// TwinCAT 3 PLC project Example
// ProgramVersion: 3.1.4026.19
// libraries:
//   Bolt, * (Zeugwerk GmbH)
//   Struckig, 0.15.5.0 (Stefan Besler)
//   Tc3_Module, * (Beckhoff Automation GmbH)
//   ZApplication, 1.5.37.1 (Zeugwerk GmbH)
//   ZAux, 1.5.37.1 (Zeugwerk GmbH)
//   ZCore, 1.5.37.1 (Zeugwerk GmbH)
//   ZEquipment, 1.5.37.1 (Zeugwerk GmbH)
//   ZPlatform, 1.5.37.1 (Zeugwerk GmbH)
// project tree:
//   ZApp/App/ ZApp.TcPOU
//   ZApp/App/_DataTypes/ ZAppStep.TcDUT
//   ZApp/App/_States/ ZAppSequenceBoot.TcPOU, ZAppSequenceBootFault.TcPOU, ZAppSequenceRunning.TcPOU
//   ZApp/App/_SubObjects/ ZAppSequence.TcPOU
//   ZApp/Com/_DataTypes/ ZCom.TcDUT (not stored), ZComUnit.TcDUT
//   ZApp/Data/_DataTypes/ ZData.TcDUT, ZDataMachine.TcDUT, ZDataConfig.TcDUT, ZDataCalibration.TcDUT (not stored), ZDataRecipe.TcDUT (not stored)
//   ZApp/Unit/Handling/ HandlingUnit.TcPOU, HandlingUnitProgram.TcPOU, IHandling.TcIO (not stored)
//   ZApp/Unit/Handling/_Com/ HandlingCom.TcDUT (not stored), HandlingComPublish.TcDUT (not stored), HandlingComPublishEquipment.TcDUT (not stored), HandlingComRef.TcDUT, HandlingComRequest.TcDUT (not stored), HandlingComSubscribe.TcDUT, HandlingComSubscribeEquipment.TcDUT (not stored)
//   ZApp/Unit/Handling/_DataTypes/ HandlingState.TcDUT, HandlingStep.TcDUT
//   ZApp/Unit/Handling/_Data/ HandlingDataCalibration.TcDUT (not stored), HandlingDataConfig.TcDUT, HandlingDataMachine.TcDUT, HandlingDataRef.TcDUT
//   ZApp/Unit/Handling/_Equipment/ HandlingActuator.TcPOU, HandlingAxis.TcPOU (not stored), HandlingCollision.TcPOU, HandlingEquipment.TcPOU (not stored), HandlingFieldbus.TcPOU (not stored), HandlingIo.TcPOU, HandlingLinkedUnit.TcPOU
//   ZApp/Unit/Handling/_States/ HandlingSequenceAutomatic.TcPOU, HandlingSequenceBoot.TcPOU, HandlingSequenceFaultReaction.TcPOU (not stored), HandlingSequenceGoHome.TcPOU (not stored), HandlingSequenceStop.TcPOU
//   ZApp/Unit/Handling/_SubObjects/ HandlingContainer.TcPOU, HandlingSequence.TcPOU
//   ZApp/Unit/Mover/ IMover.TcIO (not stored), MoverUnit.TcPOU, MoverUnitProgram.TcPOU
//   ZApp/Unit/Mover/_Com/ MoverCom.TcDUT, MoverComPublish.TcDUT (not stored), MoverComPublishEquipment.TcDUT, MoverComRef.TcDUT, MoverComRequest.TcDUT (not stored), MoverComSubscribe.TcDUT (not stored), MoverComSubscribeEquipment.TcDUT
//   ZApp/Unit/Mover/_DataTypes/ MoverState.TcDUT, MoverStep.TcDUT (not stored)
//   ZApp/Unit/Mover/_Data/ MoverDataCalibration.TcDUT (not stored), MoverDataConfig.TcDUT (not stored), MoverDataMachine.TcDUT (not stored), MoverDataRef.TcDUT
//   ZApp/Unit/Mover/_Equipment/ MoverCollision.TcPOU (not stored), MoverActuator.TcPOU, MoverAxis.TcPOU (not stored), MoverEquipment.TcPOU (not stored), MoverFieldbus.TcPOU (not stored), MoverIo.TcPOU, MoverLinkedUnit.TcPOU
//   ZApp/Unit/Mover/_States/ MoverSequenceAutomatic.TcPOU (not stored), MoverSequenceBoot.TcPOU, MoverSequenceFaultReaction.TcPOU (not stored), MoverSequenceGoHome.TcPOU (not stored), MoverSequenceStop.TcPOU (not stored)
//   ZApp/Unit/Mover/_SubObjects/ MoverContainer.TcPOU, MoverSequence.TcPOU (not stored)
//   ZApp/ ZGlobal.TcGVL (not stored), ZModuleProgram.TcPOU, ZModuleTask.TcTTO (not stored)
// real-time tasks:
//   TASK ZModuleTask: cycle T#10ms, priority 20, ADS port 350

// ---- ZApp/App/_DataTypes/ZAppStep.TcDUT
{attribute 'qualified_only'}
{attribute 'to_string'}
TYPE ZAppStep :
(
  Undefined := 0
  
  ,BootBegin
  ,BootLoadDefaultData
  ,BootEnd
  ,BootFaultBegin
  ,BootFaultEnd 
  ,RunningBegin
  ,RunningEnd   
);
END_TYPE

// ---- ZApp/Com/_DataTypes/ZComUnit.TcDUT
TYPE ZComUnit :
STRUCT
{region "Handling"}
{IF NOT (defined (Handling_disabled))}
  Handling : HandlingCom;
  {attribute 'ZId' := 'a0dd13f9-743a-4c3b-9b43-ecc916834d10'}
{END_IF}
{endregion}
{region "Mover1"}
{IF NOT (defined (Mover1_disabled))}
  Mover1 : MoverCom;
  {attribute 'ZId' := '0635b537-20e6-40de-ab4b-39921311b510'}
{END_IF}
{endregion}
{attribute '__ZwPlcApplicationComUnitDeclaration__'} // Do not remove this attribute! It is used for code generation.
END_STRUCT
END_TYPE

// ---- ZApp/Data/_DataTypes/ZData.TcDUT
TYPE ZData :
STRUCT
  Config : ZDataConfig;
  Machine : ZDataMachine;
  Calibration : ZDataCalibration;
  Recipe : ZDataRecipe;
END_STRUCT
END_TYPE

// ---- ZApp/Data/_DataTypes/ZDataMachine.TcDUT
TYPE ZDataMachine :
STRUCT
{region "Handling"}
{IF NOT (defined (Handling_disabled))}
  Handling : HandlingDataMachine;
  {attribute 'ZId' := 'a0dd13f9-743a-4c3b-9b43-ecc916834d10'}
{END_IF}
{endregion}
{region "Mover1"}
{IF NOT (defined (Mover1_disabled))}
  Mover1 : MoverDataMachine;
  {attribute 'ZId' := '0635b537-20e6-40de-ab4b-39921311b510'}
{END_IF}
{endregion}
{attribute '__ZwPlcApplicationDataMachineDeclaration__'} // Do not remove this attribute! It is used for code generation.
END_STRUCT
END_TYPE

// ---- ZApp/Data/_DataTypes/ZDataConfig.TcDUT
TYPE ZDataConfig :
STRUCT
{region "Handling"}
{IF NOT (defined (Handling_disabled))}
  Handling : HandlingDataConfig;
  {attribute 'ZId' := 'a0dd13f9-743a-4c3b-9b43-ecc916834d10'}
{END_IF}
{endregion}
{region "Mover1"}
{IF NOT (defined (Mover1_disabled))}
  Mover1 : MoverDataConfig;
  {attribute 'ZId' := '0635b537-20e6-40de-ab4b-39921311b510'}
{END_IF}
{endregion}
{attribute '__ZwPlcApplicationDataConfigDeclaration__'} // Do not remove this attribute! It is used for code generation.
END_STRUCT
END_TYPE

// ---- ZApp/Unit/Handling/_Com/HandlingComRef.TcDUT
/// container for all communication data types that are used by the unit
TYPE HandlingComRef :
STRUCT
  Publish : REFERENCE TO HandlingComPublish; 
  Subscribe : REFERENCE TO HandlingComSubscribe; 
END_STRUCT
END_TYPE

// ---- ZApp/Unit/Handling/_Com/HandlingComSubscribe.TcDUT
TYPE HandlingComSubscribe :
STRUCT
  Request : HandlingComRequest; // contains booleans that are used to start a specific sequence.
  Equipment : HandlingComSubscribeEquipment;  // structs for equipment objects which are used by the bridges
END_STRUCT
END_TYPE

// ---- ZApp/Unit/Handling/_DataTypes/HandlingState.TcDUT
/// This enumeration contains all used defined sequences of a unit.
/// Per default a unit makes use of the states that are contained in (UnitStateDefault)[xref:ZApplication.UnitStateDefault]. However,
/// most of the time a unit need to perform some application depend sequences that can be performed by putting the unit into userdefined states.
/// For instance, a robotic unit could use the state (automatic)[xref:ZApplication.UnitStateDefault] to lift an object from point A to point B,
/// a userdefined state could be used to open and close the robotic-units gripper, respectively
{attribute 'qualified_only'}
TYPE HandlingState :
(
	UserdefinedState1 := ZApplication.UnitStateMachineState.Last+1
);
END_TYPE

// ---- ZApp/Unit/Handling/_DataTypes/HandlingStep.TcDUT
/// This enumeration contains all steps that are used by the various sequences of a unit.
/// Sequences use a subrange (***Begin to ***End) of this enumeration.
{attribute 'qualified_only'}
{attribute 'to_string'}
TYPE HandlingStep :
(
  Undefined := 0
  
  ,BootBegin
  ,BootEnd 

  ,StopBegin
  ,StopEnd

  ,AutomaticBegin
  ,AutomaticSwitch
  ,AutomaticMoveInterpolatedVelocity
  ,AutomaticEnd
  
  ,GoHomeBegin
  ,GoHomeJoint3
  ,GoHomeJoint12
  ,GoHomeJoint2
  ,GoHomeEnd 
  
  ,FaultReactionBegin
  ,FaultReactionEnd
);
END_TYPE

// ---- ZApp/Unit/Handling/_Data/HandlingDataConfig.TcDUT
/// configuration data that is used during boot to configure the Units equipment
TYPE HandlingDataConfig :
STRUCT
  Simulated : BOOL;
END_STRUCT
END_TYPE

// ---- ZApp/Unit/Handling/_Data/HandlingDataMachine.TcDUT
/// machine data that is used through most sequences of the unit (motor speed, axes positions, ...)
TYPE HandlingDataMachine :
STRUCT
  Slowspeed : LREAL;
  Highspeed : LREAL;
END_STRUCT
END_TYPE

// ---- ZApp/Unit/Handling/_Data/HandlingDataRef.TcDUT
/// container for all data that are used by the unit
TYPE HandlingDataRef :
STRUCT
  Config : REFERENCE TO HandlingDataConfig; // data required for booting the unit (axes configuration, simulation, parameters that have to be written in PREOP, ...)
  Machine : REFERENCE TO HandlingDataMachine; // speeds, positions, ...
  Calibration : REFERENCE TO HandlingDataCalibration; // offsets, shifts of nominal to actual values
END_STRUCT
END_TYPE

// ---- ZApp/Unit/Mover/_Com/MoverCom.TcDUT
/// This struct contains variables that
/// * are read from outside (e.g. HMI) to retrieve information about the unit's current state and (temporary) parameters (= `publish`) 
/// * are written from outside (e.g. HMI) to control the unit via ADS (= `subscribe`) 
TYPE MoverCom :
STRUCT
  Publish : MoverComPublish;
  Subscribe : MoverComSubscribe;
END_STRUCT
END_TYPE

// ---- ZApp/Unit/Mover/_Com/MoverComPublishEquipment.TcDUT
TYPE MoverComPublishEquipment :
STRUCT

{region "AxisX : Axis"}
  AxisX : ZApplication.AxisComPublish;
  {attribute 'ZId' := '002e5115-61f4-40c1-8715-993ad81c0703'}
{endregion}

{attribute '__ZwPlcUnitComDeclaration__'} // Do not remove this attribute! It is used for code generation.

END_STRUCT
END_TYPE

// ---- ZApp/Unit/Mover/_Com/MoverComRef.TcDUT
/// container for all communication data types that are used by the unit
TYPE MoverComRef :
STRUCT
  Publish : REFERENCE TO MoverComPublish; 
  Subscribe : REFERENCE TO MoverComSubscribe; 
END_STRUCT
END_TYPE

// ---- ZApp/Unit/Mover/_Com/MoverComSubscribeEquipment.TcDUT
TYPE MoverComSubscribeEquipment :
STRUCT

{region "AxisX : Axis"}
  AxisX : ZApplication.AxisComSubscribe;
  {attribute 'ZId' := '002e5115-61f4-40c1-8715-993ad81c0703'}
{endregion}

{attribute '__ZwPlcUnitComDeclaration__'} // Do not remove this attribute! It is used for code generation.

END_STRUCT
END_TYPE

// ---- ZApp/Unit/Mover/_DataTypes/MoverState.TcDUT
/// This enumeration contains all used defined sequences of a unit.
/// Per default a unit makes use of the states that are contained in (UnitStateDefault)[xref:ZApplication.UnitStateDefault]. However,
/// most of the time a unit need to perform some application depend sequences that can be performed by putting the unit into userdefined states.
/// For instance, a robotic unit could use the state (automatic)[xref:ZApplication.UnitStateDefault] to lift an object from point A to point B,
/// a userdefined state could be used to open and close the robotic-units gripper, respectively
{attribute 'qualified_only'}
TYPE MoverState :
(
	UserdefinedState1 := ZApplication.UnitStateMachineState.Last+1
);
END_TYPE

// ---- ZApp/Unit/Mover/_Data/MoverDataRef.TcDUT
/// container for all data that are used by the unit
TYPE MoverDataRef :
STRUCT
  Config : REFERENCE TO MoverDataConfig; // data required for booting the unit (axes configuration, simulation, parameters that have to be written in PREOP, ...)
  Machine : REFERENCE TO MoverDataMachine; // speeds, positions, ...
  Calibration : REFERENCE TO MoverDataCalibration; // offsets, shifts of nominal to actual values
END_STRUCT
END_TYPE

// ---- ZApp/App/ZApp.TcPOU
FUNCTION_BLOCK ZApp EXTENDS ZApplication.Application
VAR
  _boot : ZAppSequenceBoot;
  _bootFault : ZAppSequenceBootFault;
  _running : ZAppSequenceRunning;
END_VAR

METHOD FB_init : BOOL
VAR_INPUT
  bInitRetains : BOOL; /// if TRUE, the retain variables are initialized (warm start / cold start)
  bInCopyCode : BOOL; /// if TRUE, the instance afterwards gets moved into the copy code (online change)
  displayName : ZCore.ZString;
  com : REFERENCE TO ZApplication.ApplicationComPublish;
END_VAR
SetBootSequence(_boot);
SetBootFaultSequence(_bootFault);
SetRunningSequence(_running);
END_METHOD

END_FUNCTION_BLOCK

// ---- ZApp/App/_States/ZAppSequenceBoot.TcPOU
FUNCTION_BLOCK ZAppSequenceBoot EXTENDS ZAppSequence IMPLEMENTS ZCore.ISequence
VAR
  _step : ZCore.Step(ZAppStep.BootBegin, ZAppStep.BootEnd);
END_VAR

IF OnStart(_step)
THEN
  // init custom sequence variables here ...
END_IF

REPEAT
  LogStep();

  CASE _step.Index OF
    (* -------------------------------------------------------------------------------------------------------------------------------- *)
    ZAppStep.BootBegin:
    (* -------------------------------------------------------------------------------------------------------------------------------- *)
    
      IF _step.OnEntry()
      THEN
        ZModuleProgram.LoggerFile.MinimumLevel := ZCore.LogLevel.Trace;
        ZModuleProgram.Logger.AddLogger(ZModuleProgram.LoggerFile); 
        //ZModuleProgram.World.Host := '82.165.219.190.1.1';       
        ZModuleProgram.World.SetLogger(ZModuleProgram.Logger);
        {attribute '__ZwPlcAppZComModuleContext__'} // Do not remove this attribute! It is used for code generation.      
      END_IF
      
	  IF ZModuleProgram.Datetime.State <> ZCore.ObjectState.Booting
      THEN
        _step.SetNext(ZAppStep.BootLoadDefaultData);        
      END_IF
      
    (* -------------------------------------------------------------------------------------------------------------------------------- *)
    ZAppStep.BootLoadDefaultData:
    (* -------------------------------------------------------------------------------------------------------------------------------- *)

      {warning 'The application is loading the default config data on every restart!'}
      LoadDefaultConfigData();
      
      IF IsCommissioning()
      THEN
        LoadDefaultData();
      END_IF
      
      _step.SetNext(ZAppStep.BootEnd);
      
    (* -------------------------------------------------------------------------------------------------------------------------------- *)
    ZAppStep.BootEnd:
    (* -------------------------------------------------------------------------------------------------------------------------------- *)
      SetBusy(FALSE);
      
  ELSE
    Abort('sequence contains unhandled step');
  END_CASE
UNTIL _step.IsNotRepeatable() OR_ELSE NOT Busy END_REPEAT

METHOD  IsCommissioning : BOOL
IsCommissioning := TRUE;
END_METHOD

METHOD FINAL LoadDefaultConfigData

{region "Handling"}
  {IF NOT (defined (Handling_disabled))}
  ZGlobal.Data.Config.Handling.Simulated := TRUE;
  {region "UserInitCode"}
  // put your individual init code for this unit here
  {endregion}
  {END_IF}
  {attribute 'ZId' := 'a0dd13f9-743a-4c3b-9b43-ecc916834d10'}
{endregion}

{region "Mover1"}
  {IF NOT (defined (Mover1_disabled))}
  ZGlobal.Data.Config.Mover1.Simulated := TRUE;
  {region "UserInitCode"}
  // put your individual init code for this unit here
  {endregion}
  {END_IF}
  {attribute 'ZId' := '0635b537-20e6-40de-ab4b-39921311b510'}
{endregion}

{attribute '__ZwPlcUnitLoadDefaultConfigData__'} // Do not remove this attribute! It is used for code generation.
END_METHOD

METHOD FINAL LoadDefaultData

{attribute '__ZwPlcUnitLoadDefaultData__'} // Do not remove this attribute! It is used for code generation.
END_METHOD

END_FUNCTION_BLOCK

// ---- ZApp/App/_SubObjects/ZAppSequence.TcPOU
FUNCTION_BLOCK ABSTRACT ZAppSequence EXTENDS ZApplication.Sequence IMPLEMENTS ZCore.ISequence

METHOD StepDecoded : ZCore.ZString
VAR_INPUT
  stepIndex : INT;
END_VAR
VAR_INST
  _stepIndexDecoded : ZAppStep;
END_VAR
_stepIndexDecoded := stepIndex;
StepDecoded := TO_STRING(_stepIndexDecoded);
END_METHOD

END_FUNCTION_BLOCK

// ---- ZApp/ZModuleProgram.TcPOU
/// Zeugwerk Application
PROGRAM ZModuleProgram
VAR_INPUT
{region "ZModuleProgram : Utility"}
  App : ZApp(displayName:='Zeugwerk-Application Template', com:=ZGlobal.Com.App);
  Datetime : ZAux.DateTimeUM;
  {attribute 'ZId' := ''}
{endregion}
{region "ZModuleProgram : Logging"}
  Alarming : ZApplication.Alarming(App, datetime := Datetime, com := ZGlobal.Com.Alarming);
  LoggerHmi : ZApplication.Messaging(App, datetime := Datetime, com := ZGlobal.Com.Messages);
  LoggerFile : ZAux.LoggerFile7FF(App, datetime := Datetime, filePath:='C:\Zeugwerk\logs\messages.log', target:='');
  Logger : ZAux.Logging;
  World : Bolt.CollisionWorld(App, 'E:\Bullcat\Example\world.urdf');
  {attribute 'ZId' := ''}
{endregion}  
{attribute '__ZwPlcApplicationModuleProgramDeclaration__'} // Do not remove this attribute! It is used for code generation.
{region "Handling"}
{undefine RunInSeparateProgram}
{IF NOT (defined (Handling_disabled)) AND NOT (defined (RunInSeparateProgram))}
  Handling : HandlingUnit(displayName := 'Handling', // name of the unit (for logging)
					  parent := App, // caller of the Unit's cyclic method. If the Unit runs in its own context use 0
						configdata := ZGlobal.Data.Config.Handling,
						machinedata := ZGlobal.Data.Machine.Handling,
						calibrationdata := ZGlobal.Data.Calibration.Handling,
						com := ZGlobal.Com.Unit.Handling);
  {attribute 'section' := '__ZwPlcUnitProgramDeclaration__'}
  {attribute 'ZId' := 'a0dd13f9-743a-4c3b-9b43-ecc916834d10'}
{END_IF}
{endregion}
{region "Mover1"}
{undefine RunInSeparateProgram}
{IF NOT (defined (Mover1_disabled)) AND NOT (defined (RunInSeparateProgram))}
  Mover1 : MoverUnit(displayName := 'Mover1', // name of the unit (for logging)
    parent:= App,
    configdata:= ZGlobal.Data.Config.Mover1,
    machinedata := ZGlobal.Data.Machine.Mover1,
    calibrationdata := ZGlobal.Data.Calibration.Mover1,
    com := ZGlobal.Com.Unit.Mover1,
    logger := Logger,
    alarming:= Alarming);
  {attribute 'section' := '__ZwPlcUnitProgramDeclaration__'}
  {attribute 'ZId' := '0635b537-20e6-40de-ab4b-39921311b510'}
{END_IF}
{endregion}
{attribute '__ZwPlcUnitProgramDeclaration__'} // Do not remove this attribute! It is used for code generation.
END_VAR

// do collision detection for whole machine
IF NOT World.Busy
THEN
  World.UpdateAndCheckSceneAsync();
END_IF

{region "ZModuleProgram : Utility"}
  Datetime.Cyclic();
  App.Cyclic();
  {attribute 'ZId' := ''}
{endregion}
{attribute '__ZwPlcApplicationModuleProgramImplementation__'} // Do not remove this attribute! It is used for code generation.

END_PROGRAM

// ---- ZApp/Unit/Handling/HandlingUnit.TcPOU
/// Declaration of a distinct unit of this application
FUNCTION_BLOCK HandlingUnit EXTENDS ZApplication.Unit IMPLEMENTS IHandling
VAR
  _equipment : HandlingEquipment(THIS^);
  _data : HandlingDataRef;
  _com : HandlingComRef;

  _boot : HandlingSequenceBoot(THIS^);
  _automatic : HandlingSequenceAutomatic(THIS^);
  _stop : HandlingSequenceStop(THIS^);
  _gohome : HandlingSequenceGoHome(THIS^);
  _faultReaction : HandlingSequenceFaultReaction(THIS^);
  
  _statemachine : ZApplication.UnitStateMachine;

  _observeTimer : ZAux.Timer;
END_VAR

{attribute 'ZId' := '2160a0d9-b961-4504-830a-bd7771ead3e7'}

IF _observeTimer.Done THEN
  _observeTimer.WaitAsync(0.1);
  
  // monitor _com for requested actions (e.g. start homing, start automatic mode, ...)
  ObserveRequest(_com.Subscribe.Request.Start, ZApplication.UnitStateMachineState.Automatic);
  ObserveRequest(_com.Subscribe.Request.Stop, ZApplication.UnitStateMachineState.Stop);
  ObserveRequest(_com.Subscribe.Request.GoHome, ZApplication.UnitStateMachineState.GoHome);
  ObserveRequest(_com.Subscribe.Request.Halt, ZApplication.UnitStateMachineState.Halt);
  
  // provide relevant information via ADS
  _com.Publish.Request.Stop := _stateMachine.IsTransitionAllowed(ZApplication.UnitStateMachineState.Stop);
  _com.Publish.Request.Start := _stateMachine.IsTransitionAllowed(ZApplication.UnitStateMachineState.Automatic);
  _com.Publish.Request.GoHome := _stateMachine.IsTransitionAllowed(ZApplication.UnitStateMachineState.GoHome);
  _com.Publish.Request.Halt := _stateMachine.IsTransitionAllowed(ZApplication.UnitStateMachineState.Halt);

  _com.Publish.State := _stateMachine.State();
END_IF

IF _statemachine.State() <> UnitStateMachineState.Automatic
THEN
  _equipment.Collision.Joint1.SetPosition((_equipment.Axis.Axis1.ActualPosition + _equipment.Axis.Axis1.ActualFollowingError) / 180.0 * ZCore.Constants.Pi);
  _equipment.Collision.Joint2.SetPosition((_equipment.Axis.Axis2.ActualPosition + _equipment.Axis.Axis2.ActualFollowingError) / 180.0 * ZCore.Constants.Pi);
  _equipment.Collision.Joint3.SetPosition((_equipment.Axis.Axis3.ActualPosition + _equipment.Axis.Axis3.ActualFollowingError) / 180.0 * ZCore.Constants.Pi);
END_IF

METHOD FB_init : BOOL
VAR_INPUT
  bInitRetains : BOOL; // if TRUE, the retain variables are initialized (warm start / cold start)
  bInCopyCode : BOOL;  // if TRUE, the instance afterwards gets moved into the copy code (online change)
  parent : ZCore.IManagedObject; // caller of the Unit's cyclic method. If the Unit runs in its own context use 0
  displayName : ZCore.ZString;  // name of this unit as it should show up in the logger
  configdata : REFERENCE TO HandlingDataConfig;  // reference to the configuration data that is used during boot to configure the Units equipment
  machinedata : REFERENCE TO HandlingDataMachine; // reference to the machine data that is used through most sequences of the unit (motor speed, axes positions, ...)
  calibrationdata : REFERENCE TO HandlingDataCalibration;  // reference to calibration that is determined by calibration sequences of the unit (static offsets, shifts)
  com : REFERENCE TO HandlingCom;  // reference to the communication interface that is used to control this Unit via ADS
END_VAR
_name := displayName;

// initialize local logger decorator
_loggerDecorator.FB_init(bInitRetains, bInCopyCode, _name, ZModuleProgram.Logger);
_alarmingDecorator.FB_init(bInitRetains, bInCopyCode, _name, ZModuleProgram.Alarming);

// setup data
_data.Config REF= configdata;
_data.Machine REF= machinedata;
_data.Calibration REF= calibrationdata;
_com.Publish REF= com.Publish;
_com.Subscribe REF= com.Subscribe;

// ------- sequence initialization, map sequences of this unit to the statemachine -------
{attribute '__ZwPlcUnitInitSequenceImplementation__'} // Do not remove this attribute! It is used for code generation.
_statemachine.SetSequence(ZApplication.UnitStateMachineState.Boot, _boot);
_statemachine.SetSequence(ZApplication.UnitStateMachineState.FaultReaction, _faultReaction);
_statemachine.SetSequence(ZApplication.UnitStateMachineState.Gohome, _gohome);
_statemachine.SetSequence(ZApplication.UnitStateMachineState.Stop, _stop);
_statemachine.SetSequence(ZApplication.UnitStateMachineState.Automatic, _automatic);

_statemachine.SetName(_name);
_statemachine.SetLogger(_logger);

// set initial state
_statemachine.SetState(ZApplication.UnitStateMachineState.Boot);
SetStateMachine(_statemachine);
END_METHOD

END_FUNCTION_BLOCK

// ---- ZApp/Unit/Handling/_States/HandlingSequenceBoot.TcPOU
FUNCTION_BLOCK HandlingSequenceBoot EXTENDS HandlingSequence IMPLEMENTS ZCore.ISequence
VAR
  _step : ZCore.Step(HandlingStep.BootBegin, HandlingStep.BootEnd);
END_VAR

IF OnStart(_step) THEN
  ; // init custom sequence variables here ...
END_IF

REPEAT
  LogStep();

  CASE _step.Index OF
    (* -------------------------------------------------------------------------------------------------------------------------------- *)
    HandlingStep.BootBegin:
    (* -------------------------------------------------------------------------------------------------------------------------------- *)
      IF _step.OnEntry()
      THEN
        // initialize equipment
        _io();
        _actuator();
        _fieldbus();
        _axis();
        _collision();
        _unit();
      END_IF
      
      _parent._objectManager.Cyclic();      
      Assert(_parent._objectManager);
      IF _parent._objectManager.Booted
      THEN
        _step.SetNext(HandlingStep.BootEnd);
      END_IF

    (* -------------------------------------------------------------------------------------------------------------------------------- *)
    HandlingStep.BootEnd:
    (* -------------------------------------------------------------------------------------------------------------------------------- *)
      SetBusy(FALSE);
      
  ELSE
    Abort('sequence contains unhandled step');
  END_CASE
UNTIL _step.IsNotRepeatable() OR_ELSE NOT Busy END_REPEAT

END_FUNCTION_BLOCK

// ---- ZApp/Unit/Handling/_SubObjects/HandlingSequence.TcPOU
FUNCTION_BLOCK HandlingSequence EXTENDS ZApplication.Sequence
VAR
  {attribute 'hide'}
  _parent : REFERENCE TO HandlingUnit;
  _io : REFERENCE TO HandlingIo;
  _actuator : REFERENCE TO HandlingActuator;
  _fieldbus : REFERENCE TO HandlingFieldbus;
  _axis : REFERENCE TO HandlingAxis;
  _collision : REFERENCE TO HandlingCollision;  
  _data : REFERENCE TO HandlingDataRef;
  _unit : REFERENCE TO HandlingLinkedUnit;  
END_VAR

METHOD FB_init : BOOL
VAR_INPUT
  bInitRetains : BOOL; // if TRUE, the retain variables are initialized (warm start / cold start)
  bInCopyCode : BOOL;  // if TRUE, the instance afterwards gets moved into the copy code (online change)
  unit : REFERENCE TO HandlingUnit;
END_VAR
_parent REF= unit;
_alarming := unit._alarming;
_io REF= unit._equipment.Io;
_actuator REF= unit._equipment.Actuator;
_fieldbus REF= unit._equipment.Fieldbus;
_axis REF= unit._equipment.Axis;
_collision REF= unit._equipment.Collision;
_unit REF= unit._equipment.Unit;
_data REF= unit._data;
_loggerDiagnostics.SetLogger(unit._logger);
END_METHOD

METHOD StepDecoded : ZCore.ZString
VAR_INPUT
  stepIndex : INT;
END_VAR
VAR_INST
  _stepIndexDecoded : HandlingStep;
END_VAR
_stepIndexDecoded := stepIndex;
stepDecoded := TO_STRING(_stepIndexDecoded);
END_METHOD

END_FUNCTION_BLOCK

// ---- ZApp/Unit/Handling/_Equipment/HandlingIo.TcPOU
/// This function block is a container for all I/Os that are used by this unit.
/// The parent of all objects can be directly transfered in their constructor (this is only relevant for equipment objects
/// that have to be managed (e.g. [DebouncedInput](xref:ZEquipment.DebouncedInput), [Light](xref:ZEquipment.Light), ...).
FUNCTION_BLOCK HandlingIo EXTENDS HandlingContainer
VAR
  {attribute 'hide'}
  _iobridge : ZApplication.IoBridge(_parent);
END_VAR
VAR_INPUT

{attribute '__ZwPlcUnitEquipmentDeclaration__'} // Do not remove this attribute! It is used for code generation.
END_VAR

IF _isInitialized
THEN
  RETURN;
END_IF

  _iobridge.SetLogger(_parent._logger);

{attribute '__ZwPlcUnitEquipmentImplementation__'} // Do not remove this attribute! It is used for code generation.

_isInitialized := TRUE;

END_FUNCTION_BLOCK

// ---- ZApp/Unit/Handling/_SubObjects/HandlingContainer.TcPOU
FUNCTION_BLOCK HandlingContainer EXTENDS ZCore.ObjectContainer
VAR_INPUT
END_VAR
VAR_OUTPUT
END_VAR
VAR
  {attribute 'hide'}
  _parent : REFERENCE TO HandlingUnit;
END_VAR

{attribute 'hide' }
METHOD FB_init : BOOL
VAR_INPUT
	bInitRetains : BOOL; // if TRUE, the retain variables are initialized (warm start / cold start)
	bInCopyCode : BOOL;  // if TRUE, the instance afterwards gets moved into the copy code (online change)
  unit : REFERENCE TO HandlingUnit;
END_VAR
_parent REF= unit;
END_METHOD

END_FUNCTION_BLOCK

// ---- ZApp/Unit/Handling/_Equipment/HandlingActuator.TcPOU
/// This function block is a container for all actuator objects that are used by this unit.
/// The parent of all objects can be directly transfered in their constructor (this is only relevant for equipment objects
/// that have to be managed (e.g. [DebouncedInput](xref:ZEquipment.DebouncedInput), [Light](xref:ZEquipment.Light), ...).
FUNCTION_BLOCK HandlingActuator EXTENDS HandlingContainer
VAR
  {attribute 'hide'}
  _actuatorbridge : ZApplication.ActuatorBridge(_parent);
  {attribute 'hide'}
  _iobridge : ZApplication.IoBridge(_parent);
END_VAR
VAR_INPUT

{attribute '__ZwPlcUnitEquipmentDeclaration__'} // Do not remove this attribute! It is used for code generation.
END_VAR

IF _isInitialized
THEN
  RETURN;
END_IF

  _actuatorbridge.SetLogger(_parent._logger);

{attribute '__ZwPlcUnitEquipmentImplementation__'} // Do not remove this attribute! It is used for code generation.

_isInitialized := TRUE;

END_FUNCTION_BLOCK

// ---- ZApp/Unit/Handling/_Equipment/HandlingCollision.TcPOU
/// This function block is a container for all axis objects that are used by this unit.
/// The parent of all objects can be directly transfered in their constructor (this is only relevant for equipment objects
/// that have to be managed (e.g. [DebouncedInput](xref:ZEquipment.DebouncedInput), [Light](xref:ZEquipment.Light), ...).
FUNCTION_BLOCK HandlingCollision EXTENDS HandlingContainer
VAR
  {attribute 'hide'}
  _axisbridge : ZApplication.AxisBridge(_parent);
END_VAR
VAR_INPUT
  World : REFERENCE TO Bolt.CollisionWorld;
  Joint1 : Bolt.Joint('joint1', ZModuleProgram.World);
  Joint2 : Bolt.Joint('joint2', ZModuleProgram.World);
  Joint3 : Bolt.Joint('joint3', ZModuleProgram.World);
END_VAR

IF _isInitialized
THEN
  RETURN;
END_IF

World REF= ZModuleProgram.World;
Joint1.SetCollisionFilter(group := 1, mask := 2#11111101);
Joint2.SetCollisionFilter(group := 1, mask := 2#11111101);
Joint3.SetCollisionFilter(group := 1, mask := 2#11111101);

_isInitialized := TRUE;

END_FUNCTION_BLOCK

// ---- ZApp/Unit/Handling/_Equipment/HandlingLinkedUnit.TcPOU
/// This function block is a container for all linked units that are used by this unit.
/// Linked units can be addressed through their individual interface.
FUNCTION_BLOCK HandlingLinkedUnit EXTENDS HandlingContainer
VAR_INPUT

{attribute '__ZwPlcUnitEquipmentDeclaration__'} // Do not remove this attribute! It is used for code generation.
END_VAR

IF _isInitialized
THEN
  RETURN;
END_IF

{attribute '__ZwPlcUnitEquipmentImplementation__'} // Do not remove this attribute! It is used for code generation.

_isInitialized := TRUE;

END_FUNCTION_BLOCK

// ---- ZApp/Unit/Handling/_States/HandlingSequenceAutomatic.TcPOU
FUNCTION_BLOCK HandlingSequenceAutomatic EXTENDS HandlingSequence IMPLEMENTS ZCore.ISequence
VAR
  _step : ZCore.Step(HandlingStep.AutomaticBegin, HandlingStep.AutomaticEnd);
  _avoidance : BOOL := TRUE;
  _rt : ZAux.RealTime;
  _otg : Struckig.Otg(0.010, 1);  
  _pid : Pid(0.010);
  _kp : LREAL := 3100;
  _ki : LREAL := 2000;
  _kd : LREAL := 0;
  
  _distance, _tableDistance : LREAL;
END_VAR

IF NOT Busy THEN
  RETURN;
END_IF

IF OnStart(_step) THEN
  ; // init custom sequence variables here ...
END_IF

IF OnStop() THEN
  RETURN; // external stop was triggered
END_IF

IF OnHalt() THEN
  ; // Halting := TRUE; // Uncomment to acknowledge that the sequence is halting
END_IF

REPEAT
  LogStep();

  CASE _step.Index OF
    (* -------------------------------------------------------------------------------------------------------------------------------- *)
    HandlingStep.AutomaticBegin:
    (* -------------------------------------------------------------------------------------------------------------------------------- *)
      IF _step.OnEntry()
      THEN
        _axis.Axis1.MoveVelocityAsync(THIS^, 50);
		    _axis.Axis2.MoveAbsoluteAsync(THIS^, 60, 50);
		    _axis.Axis3.MoveAbsoluteAsync(THIS^, 60, 50);
      END_IF

      IF _avoidance
      THEN
        Await2(obj1:=_axis.Axis2, obj2:=_axis.Axis3, nextStep:=HandlingStep.AutomaticSwitch);  
      END_IF
      
    (* -------------------------------------------------------------------------------------------------------------------------------- *)
    HandlingStep.AutomaticSwitch:
    (* -------------------------------------------------------------------------------------------------------------------------------- *)
      IF _step.OnEntry()
      THEN
        _axis.Axis2.MoveInterpolatedVelocityAsync(THIS^);
      END_IF

      Await(obj1:=_axis.Axis2, nextStep:=HandlingStep.AutomaticMoveInterpolatedVelocity);  
    
    (* -------------------------------------------------------------------------------------------------------------------------------- *)
    HandlingStep.AutomaticMoveInterpolatedVelocity:
    (* -------------------------------------------------------------------------------------------------------------------------------- *)
      IF _step.OnEntry()
      THEN
        _otg.CycleTime := _rt.CycleTimeInSeconds();
        _otg.ControlInterface := Struckig.ControlInterfaceType.Velocity;
        _otg.Discretization := Struckig.DiscretizationType.Discrete;
        _otg.EnableAutoPropagate := TRUE;  
        _otg.Synchronization := Struckig.SynchronizationType.Phase;        
        _otg.MaxJerk[0] := 100000;
        _otg.MaxAcceleration[0] := 10000;
        _otg.MaxVelocity[0] := 100;
        
        _otg.CurrentPosition[0] := _axis.Axis2.ActualPosition + _axis.Axis2.ActualFollowingError;
        _otg.CurrentVelocity[0] := 0;
        _otg.CurrentAcceleration[0] := 0;
        _otg.TargetPosition[0] := 0; 
        _otg.TargetVelocity[0] := 0; 
        _otg.TargetAcceleration[0] := 0; 
        
        _otg();
        
        _pid.SetCycleTime(_rt.CycleTimeInSeconds());
        _pid.SetControllerParametersParallel(_kp, _ki, _kd);
        _pid.SetAntiWindupType(ZCore.PidAntiWindupType.ConditionalClamping);
        _pid.SetSetPoint(00.05);
        _pid.EnableAntiWindup(TRUE, -100, 100);
      
      ELSE
        _tableDistance := _collision.World.FindMinimumDistanceByName('table');
        _distance := MIN(_collision.World.FindMinimumDistanceByName('ee_link'), MIN(_collision.World.FindMinimumDistanceByName('link2'), _tableDistance));
        _pid.SetInput(_distance);
        
        _pid.Cyclic();
        _otg.TargetVelocity[0] := -_pid.Output();
      END_IF  
    
    (* -------------------------------------------------------------------------------------------------------------------------------- *)
    HandlingStep.AutomaticEnd:
    (* -------------------------------------------------------------------------------------------------------------------------------- *)
      SetBusy(FALSE);
  
  ELSE
    Abort('sequence contains unhandled step');
  END_CASE
UNTIL _step.IsNotRepeatable() OR_ELSE NOT Busy END_REPEAT


IF _step.Index >= HandlingStep.AutomaticMoveInterpolatedVelocity
THEN
  _otg();
  
  IF _otg.State = Struckig.TrajectoryState.Error
  THEN
    Abort(_otg.ErrorMessage());
  ELSE
    _axis.Axis2.SetInterpolatedVelocity(THIS^, _otg.CurrentVelocity[0]);
    
    _collision.Joint1.SetPosition((_axis.Axis1.ActualPosition + _axis.Axis1.ActualFollowingError) / 180.0 * ZCore.Constants.Pi);
    _collision.Joint2.SetPosition((_axis.Axis2.ActualPosition + _axis.Axis2.ActualFollowingError) / 180.0 * ZCore.Constants.Pi);    
    _collision.Joint2.SetPosition((_otg.CurrentPosition[0]) / 180.0 * ZCore.Constants.Pi); // needed for simulation
    _collision.Joint3.SetPosition((_axis.Axis3.ActualPosition + _axis.Axis3.ActualFollowingError) / 180.0 * ZCore.Constants.Pi);    
	END_IF

END_IF

END_FUNCTION_BLOCK

// ---- ZApp/Unit/Handling/_States/HandlingSequenceStop.TcPOU
FUNCTION_BLOCK HandlingSequenceStop EXTENDS HandlingSequence IMPLEMENTS ZCore.ISequence
VAR
  _step : ZCore.Step(HandlingStep.StopBegin, HandlingStep.StopEnd);
  _timerSim : ZAux.Timer;
END_VAR

IF OnStart(_step) THEN
  ; // init custom sequence variables here ...
END_IF

REPEAT
  LogStep();

  CASE _step.Index OF
    (* -------------------------------------------------------------------------------------------------------------------------------- *)
    HandlingStep.StopBegin:
    (* -------------------------------------------------------------------------------------------------------------------------------- *)
      IF _step.OnEntry()
      THEN
        _timerSim.WaitAsync(5);
			END_IF
      
      Await(_timerSim, nextStep:=HandlingStep.StopEnd);
      // _step.SetNext(index:=HandlingStep.StopEnd);

    (* -------------------------------------------------------------------------------------------------------------------------------- *)
    HandlingStep.StopEnd:
    (* -------------------------------------------------------------------------------------------------------------------------------- *)    
      SetBusy(FALSE);
  
  ELSE
    Abort('sequence contains unhandled step');
  END_CASE
UNTIL _step.IsNotRepeatable() OR_ELSE NOT Busy END_REPEAT

END_FUNCTION_BLOCK

// ---- ZApp/Unit/Mover/MoverUnit.TcPOU
FUNCTION_BLOCK MoverUnit EXTENDS ZApplication.Unit IMPLEMENTS IMover
VAR
  _equipment : MoverEquipment(THIS^);
  _data : MoverDataRef;
  _com : MoverComRef;

  _boot : MoverSequenceBoot(THIS^);
  _automatic : MoverSequenceAutomatic(THIS^);
  _stop : MoverSequenceStop(THIS^);
  _gohome : MoverSequenceGoHome(THIS^);
  _faultReaction : MoverSequenceFaultReaction(THIS^);
  
  _statemachine : ZApplication.UnitStateMachine;

  _observeTimer : ZAux.Timer;
END_VAR

{attribute 'ZId' := '673a347d-1adf-4db2-ba4b-4b1c8ade11cf'}

_equipment.Collision.Box.SetPosition(1.45 + (_equipment.Axis.AxisX.ActualPosition + _equipment.Axis.AxisX.ActualFollowingError), 0.02, 0.05);

IF _observeTimer.Done THEN
  _observeTimer.WaitAsync(0.1);
  
  // monitor _com for requested actions (e.g. start homing, start automatic mode, ...)
  ObserveRequest(_com.Subscribe.Request.Start, ZApplication.UnitStateMachineState.Automatic);
  ObserveRequest(_com.Subscribe.Request.Stop, ZApplication.UnitStateMachineState.Stop);
  ObserveRequest(_com.Subscribe.Request.GoHome, ZApplication.UnitStateMachineState.GoHome);
  ObserveRequest(_com.Subscribe.Request.Halt, ZApplication.UnitStateMachineState.Halt);
  
  // provide relevant information via ADS
  _com.Publish.Request.Stop := _stateMachine.IsTransitionAllowed(ZApplication.UnitStateMachineState.Stop);
  _com.Publish.Request.Start := _stateMachine.IsTransitionAllowed(ZApplication.UnitStateMachineState.Automatic);
  _com.Publish.Request.GoHome := _stateMachine.IsTransitionAllowed(ZApplication.UnitStateMachineState.GoHome);
  _com.Publish.Request.Halt := _stateMachine.IsTransitionAllowed(ZApplication.UnitStateMachineState.Halt);

  _com.Publish.State := _stateMachine.State();
END_IF

METHOD FB_init : BOOL
VAR_INPUT
  bInitRetains : BOOL;
  bInCopyCode : BOOL;
  parent : ZCore.IManagedObject;
  displayName : ZCore.ZString;
  configdata : REFERENCE TO MoverDataConfig;
  machinedata : REFERENCE TO MoverDataMachine;
  calibrationdata : REFERENCE TO MoverDataCalibration;
  com : REFERENCE TO MoverCom;
  logger : ZCore.ILogger;
  alarming: ZApplication.IAlarming;
END_VAR
_name := displayName;

// initialize local logger decorator
_loggerDecorator.FB_init(bInitRetains, bInCopyCode, _name, logger);
_alarmingDecorator.FB_init(bInitRetains, bInCopyCode, _name, alarming);

// setup data
_data.Config REF= configdata;
_data.Machine REF= machinedata;
_data.Calibration REF= calibrationdata;
_com.Publish REF= com.Publish;
_com.Subscribe REF= com.Subscribe;

// ------- sequence initialization, map sequences of this unit to the statemachine -------
{attribute '__ZwPlcUnitInitSequenceImplementation__'} // Do not remove this attribute! It is used for code generation.
_statemachine.SetSequence(ZApplication.UnitStateMachineState.Boot, _boot);
_statemachine.SetSequence(ZApplication.UnitStateMachineState.FaultReaction, _faultReaction);
_statemachine.SetSequence(ZApplication.UnitStateMachineState.Gohome, _gohome);
_statemachine.SetSequence(ZApplication.UnitStateMachineState.Stop, _stop);
_statemachine.SetSequence(ZApplication.UnitStateMachineState.Automatic, _automatic);

_statemachine.SetName(_name);
_statemachine.SetLogger(_logger);

// set initial state
_statemachine.SetState(ZApplication.UnitStateMachineState.Boot);
SetStateMachine(_statemachine);
END_METHOD

END_FUNCTION_BLOCK

// ---- ZApp/Unit/Mover/_States/MoverSequenceBoot.TcPOU
FUNCTION_BLOCK MoverSequenceBoot EXTENDS MoverSequence IMPLEMENTS ZCore.ISequence
VAR
  _step : ZCore.Step(MoverStep.BootBegin, MoverStep.BootEnd);
END_VAR

IF OnStart(_step) THEN
  ; // init custom sequence variables here ...
END_IF

REPEAT
  LogStep();

  CASE _step.Index OF
    (* -------------------------------------------------------------------------------------------------------------------------------- *)
    MoverStep.BootBegin:
    (* -------------------------------------------------------------------------------------------------------------------------------- *)
      IF _step.OnEntry()
      THEN
        // initialize equipment
        _io();
        _actuator();
        _collision();
        _fieldbus();
        _axis();
        _unit();
      END_IF
      
      _parent._objectManager.Cyclic();      
      Assert(_parent._objectManager);
      IF _parent._objectManager.Booted
      THEN
        _step.SetNext(MoverStep.BootEnd);
      END_IF

    (* -------------------------------------------------------------------------------------------------------------------------------- *)
    MoverStep.BootEnd:
    (* -------------------------------------------------------------------------------------------------------------------------------- *)
      SetBusy(FALSE);
      
  ELSE
    Abort('sequence contains unhandled step');
  END_CASE
UNTIL _step.IsNotRepeatable() OR_ELSE NOT Busy END_REPEAT

END_FUNCTION_BLOCK

// ---- ZApp/App/_States/ZAppSequenceBootFault.TcPOU
FUNCTION_BLOCK ZAppSequenceBootFault EXTENDS ZAppSequence IMPLEMENTS ZCore.ISequence
VAR
  _step : ZCore.Step(ZAppStep.BootFaultBegin, ZAppStep.BootFaultEnd);
END_VAR

IF OnStart(_step)
THEN
  // init custom sequence variables here ...
END_IF

REPEAT
  LogStep();

  CASE _step.Index OF
    (* -------------------------------------------------------------------------------------------------------------------------------- *)
    ZAppStep.BootFaultBegin:
    (* -------------------------------------------------------------------------------------------------------------------------------- *)
      _step.SetNext(ZAppStep.BootFaultEnd);
      
    (* -------------------------------------------------------------------------------------------------------------------------------- *)
    ZAppStep.BootFaultEnd:
    (* -------------------------------------------------------------------------------------------------------------------------------- *)
      SetBusy(FALSE);
      
  ELSE
    Abort('sequence contains unhandled step');
  END_CASE
UNTIL _step.IsNotRepeatable() OR_ELSE NOT Busy END_REPEAT

END_FUNCTION_BLOCK

// ---- ZApp/App/_States/ZAppSequenceRunning.TcPOU
FUNCTION_BLOCK ZAppSequenceRunning EXTENDS ZAppSequence IMPLEMENTS ZCore.ISequence
VAR
  _step : ZCore.Step(ZAppStep.RunningBegin, ZAppStep.RunningEnd);
END_VAR

IF OnStart(_step)
THEN
  // init custom sequence variables here ...
END_IF

REPEAT
  LogStep();

  CASE _step.Index OF
    (* -------------------------------------------------------------------------------------------------------------------------------- *)
    ZAppStep.RunningBegin:
    (* -------------------------------------------------------------------------------------------------------------------------------- *)
      ; // implement me
      
    (* -------------------------------------------------------------------------------------------------------------------------------- *)
    ZAppStep.RunningEnd:
    (* -------------------------------------------------------------------------------------------------------------------------------- *)
      SetBusy(FALSE);
      
  ELSE
    Abort('sequence contains unhandled step');
  END_CASE
UNTIL _step.IsNotRepeatable() OR_ELSE NOT Busy END_REPEAT

END_FUNCTION_BLOCK

// ---- ZApp/Unit/Handling/HandlingUnitProgram.TcPOU
/// each unit can run in its own PROGRAM and Task, respectively. However, this is optional and one may also
/// instantiate the unit in the ModuleProgram.
/// In order to keep initialization to a minimum, all ModuleContext objects that are required by the Unit are
/// given as FB_init parameter. These objects are
/// * data structs
/// * communication structs
/// * busmaster(s)
/// A unit should always be a root object (no parent) if it is running in its own context. If it runs in the same
/// task as the Module the parent may be set to the Module's Application.
PROGRAM HandlingUnitProgram
VAR
{region "Handling"}
{undefine RunInSeparateProgram}
{IF NOT (defined (Handling_disabled)) AND (defined (RunInSeparateProgram))}
  Handling : HandlingUnit(displayName := 'Handling', // name of the unit (for logging)
					  parent := 0, // caller of the Unit's cyclic method. If the Unit runs in its own context use 0
						configdata := ZGlobal.Data.Config.Handling,
						machinedata := ZGlobal.Data.Machine.Handling,
						calibrationdata := ZGlobal.Data.Calibration.Handling,
						com := ZGlobal.Com.Unit.Handling);
  {attribute 'section' := '__ZwPlcUnitProgramDeclaration__'}
  {attribute 'ZId' := 'a0dd13f9-743a-4c3b-9b43-ecc916834d10'}
{END_IF}
{endregion}
{attribute '__ZwPlcUnitProgramDeclaration__'} // Do not remove this attribute! It is used for code generation.
END_VAR

// run the unit - the cylics of all children will be called as well

{region "Handling"}
{undefine RunInSeparateProgram}
{IF NOT (defined (Handling_disabled)) AND (defined (RunInSeparateProgram))}
  Handling.Cyclic();
  {attribute 'section' := '__ZwPlcUnitProgramImplementation__'}
  {attribute 'ZId' := 'a0dd13f9-743a-4c3b-9b43-ecc916834d10'}
{END_IF}
{endregion}
{attribute '__ZwPlcUnitProgramImplementation__'} // Do not remove this attribute! It is used for code generation.

END_PROGRAM

// ---- ZApp/Unit/Mover/MoverUnitProgram.TcPOU
/// each unit can run in its own PROGRAM and Task, respectively. However, this is optional and one may also
/// instantiate the unit in the ModuleProgram.
/// In order to keep initialization to a minimum, all ModuleContext objects that are required by the Unit are
/// given as FB_init parameter. These objects are
/// * data structs
/// * communication structs
/// * busmaster(s)
/// A unit should always be a root object (no parent) if it is running in its own context. If it runs in the same
/// task as the Module the parent may be set to the Module's Application.
PROGRAM MoverUnitProgram
VAR
{region "Mover1"}
{undefine RunInSeparateProgram}
{IF NOT (defined (Mover1_disabled)) AND (defined (RunInSeparateProgram))}
  Mover1 : MoverUnit(displayName := 'Mover1', // name of the unit (for logging)
    parent:= 0,
    configdata := ZGlobal.Data.Config.Mover1,
    machinedata := ZGlobal.Data.Machine.Mover1,
    calibrationdata := ZGlobal.Data.Calibration.Mover1,
    com := ZGlobal.Com.Unit.Mover1,
    logger := Logger,
    alarming:= Alarming);
  {attribute 'section' := '__ZwPlcUnitProgramDeclaration__'}
  {attribute 'ZId' := '0635b537-20e6-40de-ab4b-39921311b510'}
{END_IF}
{endregion}
{attribute '__ZwPlcUnitProgramDeclaration__'} // Do not remove this attribute! It is used for code generation.
END_VAR

// run the unit - the cylics of all children will be called as well

{region "Mover1"}
{undefine RunInSeparateProgram}
{IF NOT (defined (Mover1_disabled)) AND (defined (RunInSeparateProgram))}
  Mover1.Cyclic();
  {attribute 'section' := '__ZwPlcUnitProgramImplementation__'}
  {attribute 'ZId' := '0635b537-20e6-40de-ab4b-39921311b510'}
{END_IF}
{endregion}
{attribute '__ZwPlcUnitProgramImplementation__'} // Do not remove this attribute! It is used for code generation.

END_PROGRAM

// ---- ZApp/Unit/Mover/_Equipment/MoverActuator.TcPOU
/// This function block is a container for all actuator objects that are used by this unit.
/// The parent of all objects can be directly transfered in their constructor (this is only relevant for equipment objects
/// that have to be managed (e.g. [DebouncedInput](xref:ZEquipment.DebouncedInput), [Light](xref:ZEquipment.Light), ...).
FUNCTION_BLOCK MoverActuator EXTENDS MoverContainer
VAR
  {attribute 'hide'}
  _actuatorbridge : ZApplication.ActuatorBridge(_parent);
  {attribute 'hide'}
  _iobridge : ZApplication.IoBridge(_parent);
END_VAR
VAR_INPUT

{attribute '__ZwPlcUnitEquipmentDeclaration__'} // Do not remove this attribute! It is used for code generation.
END_VAR

IF _isInitialized
THEN
  RETURN;
END_IF

  _actuatorbridge.SetLogger(_parent._logger);

{attribute '__ZwPlcUnitEquipmentImplementation__'} // Do not remove this attribute! It is used for code generation.

_isInitialized := TRUE;

END_FUNCTION_BLOCK

// ---- ZApp/Unit/Mover/_SubObjects/MoverContainer.TcPOU
FUNCTION_BLOCK MoverContainer EXTENDS ZCore.ObjectContainer
VAR_INPUT
END_VAR
VAR_OUTPUT
END_VAR
VAR
  {attribute 'hide'}
  _parent : REFERENCE TO MoverUnit;
END_VAR

{attribute 'hide' }
METHOD FB_init : BOOL
VAR_INPUT
	bInitRetains : BOOL; // if TRUE, the retain variables are initialized (warm start / cold start)
	bInCopyCode : BOOL;  // if TRUE, the instance afterwards gets moved into the copy code (online change)
  unit : REFERENCE TO MoverUnit;
END_VAR
_parent REF= unit;
END_METHOD

END_FUNCTION_BLOCK

// ---- ZApp/Unit/Mover/_Equipment/MoverIo.TcPOU
/// This function block is a container for all I/Os that are used by this unit.
/// The parent of all objects can be directly transfered in their constructor (this is only relevant for equipment objects
/// that have to be managed (e.g. [DebouncedInput](xref:ZEquipment.DebouncedInput), [Light](xref:ZEquipment.Light), ...).
FUNCTION_BLOCK MoverIo EXTENDS MoverContainer
VAR
  {attribute 'hide'}
  _iobridge : ZApplication.IoBridge(_parent);
END_VAR
VAR_INPUT

{attribute '__ZwPlcUnitEquipmentDeclaration__'} // Do not remove this attribute! It is used for code generation.
END_VAR

IF _isInitialized
THEN
  RETURN;
END_IF

  _iobridge.SetLogger(_parent._logger);

{attribute '__ZwPlcUnitEquipmentImplementation__'} // Do not remove this attribute! It is used for code generation.

_isInitialized := TRUE;

END_FUNCTION_BLOCK

// ---- ZApp/Unit/Mover/_Equipment/MoverLinkedUnit.TcPOU
/// This function block is a container for all linked units that are used by this unit.
/// Linked units can be addressed through their individual interface.
FUNCTION_BLOCK MoverLinkedUnit EXTENDS MoverContainer
VAR_INPUT

{attribute '__ZwPlcUnitEquipmentDeclaration__'} // Do not remove this attribute! It is used for code generation.
END_VAR

IF _isInitialized
THEN
  RETURN;
END_IF

{attribute '__ZwPlcUnitEquipmentImplementation__'} // Do not remove this attribute! It is used for code generation.

_isInitialized := TRUE;

END_FUNCTION_BLOCK
